FUNCTION_BLOCK FBWriteString
VAR_INPUT
	sNetID			: STRING;
	sPath			: STRING;
	sSaveStrng		: STRING(255);
	bWrite			: BOOL;
END_VAR

VAR_OUTPUT
	bBusy			: BOOL;
	bDone			: BOOL;
	bError			: BOOL;
	iErrorID			: INT;
END_VAR

VAR
	iWrtState			: INT;
	fbR_TRIG		: R_TRIG;
	fbFB_FileOpen		: FB_FileOpen;
	fbFB_FilePuts		: FB_FilePuts;
	fbFB_FileClose		: FB_FileClose;
END_VAR

(* call FB's *)
fileFBs();
fbR_TRIG(CLK:=bWrite, Q=> );

CASE iWrtState OF
0:	(* idle *)
	IF fbR_TRIG.Q THEN
		iWrtState:=10;
		bBusy:=TRUE;
		bError:=FALSE;
		iErrorID:=0;
	END_IF
	IF NOT(bWrite) THEN
		bDone:=FALSE;
	END_IF

10:
	(* File Open *)	(* ==> could leave file open for faster performance?? *)
	(* when busy bit goes false, if no error, then should have successfully opened file *)
	IF NOT(fbFB_FileOpen.bBusy) AND NOT(fbFB_FileOpen.bError) THEN
		iWrtState:=20;
	END_IF

	IF fbFB_FileOpen.bError THEN
		iWrtState:=101;
	END_IF

20:
	(* File Write *)
	(* when busy bit goes false, if no error, then should have successfully written to file *)
	IF NOT(fbFB_FilePuts.bBusy) AND NOT(fbFB_FilePuts.bError) THEN
		iWrtState:=30;
	END_IF

	IF fbFB_FilePuts.bError THEN
		iWrtState:=102;
	END_IF

30:
	(* File Close *)
	(* when busy bit goes false, if no error, then should have successfully closed file *)
	IF NOT(fbFB_FileClose.bBusy) AND NOT(fbFB_FileClose.bError) THEN
		iWrtState:=40;
	END_IF

	IF fbFB_FileClose.bError THEN
		iWrtState:=103;
	END_IF

40:
	(* Write to file complete -- return to idle state *)
	iWrtState:=0;
	bDone:=TRUE;
	bBusy:=FALSE;

101:	(* open error handler *)
	bError:=TRUE;
	bBusy:=FALSE;
	iErrorID:=iWrtState;
	iWrtState:=0;

102:	(* write error handler *)
	bError:=TRUE;
	bBusy:=FALSE;
	iErrorID:=iWrtState;
	iWrtState:=0;

103:	(* close error handler *)
	bError:=TRUE;
	bBusy:=FALSE;
	iErrorID:=iWrtState;
	iWrtState:=0;

END_CASE

ACTION FileFBs:
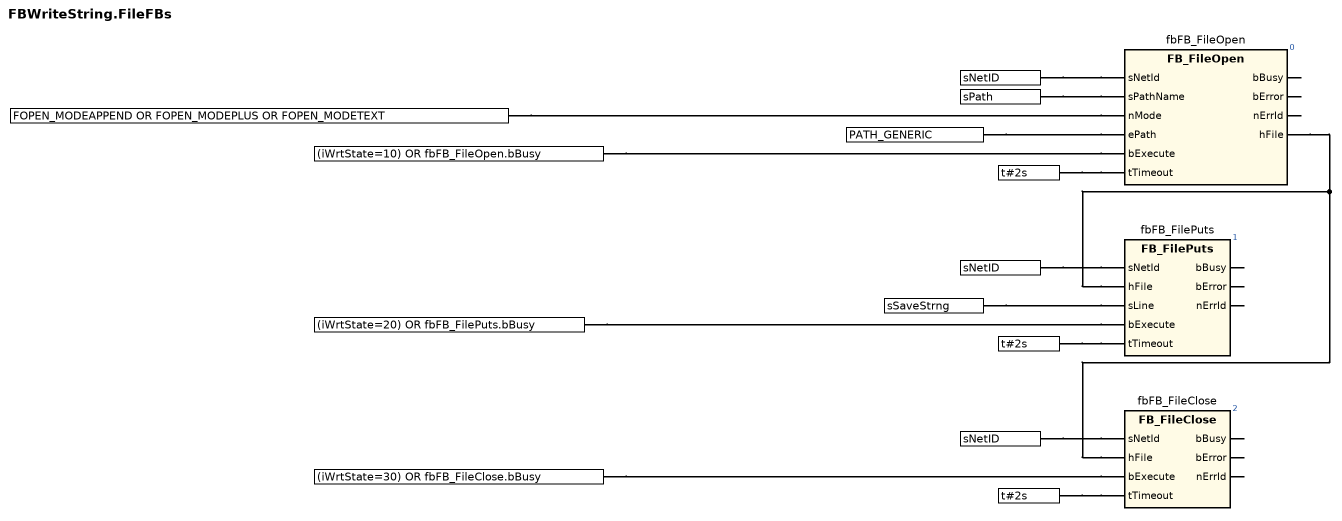
fbFB_FileOpen(
    sNetId := sNetID,
    sPathName := sPath,
    nMode := FOPEN_MODEAPPEND OR FOPEN_MODEPLUS OR FOPEN_MODETEXT,
    ePath := PATH_GENERIC,
    bExecute := (iWrtState=10) OR fbFB_FileOpen.bBusy,
    tTimeout := t#2s); // FB_FileOpen
fbFB_FilePuts(
    sNetId := sNetID,
    hFile := fbFB_FileOpen.hFile,
    sLine := sSaveStrng,
    bExecute := (iWrtState=20) OR fbFB_FilePuts.bBusy,
    tTimeout := t#2s); // FB_FilePuts
fbFB_FileClose(
    sNetId := sNetID,
    hFile := fbFB_FileOpen.hFile,
    bExecute := (iWrtState=30) OR fbFB_FileClose.bBusy,
    tTimeout := t#2s); // FB_FileClose
END_ACTION

END_FUNCTION_BLOCK

(* stored: Version 1.1.0.1, ProductVersion 3.1.4018.5
   POU FBWriteString: Id {ddb88e17-e597-4798-b003-6932acf98330}, SpecialFunc None
   Action FileFBs: Id {ed642076-748a-4bb3-af88-f9a279d7c153} *)
